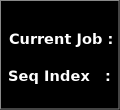
VISUALIZATION PUSeq  // 120x110
    Rectangle (0,0 371x118)
        OnMouseDown: CloseDialog Dialog=PUSeq, Result=None, NumpadKeypadSet=True
    Label (6,24 114x30), "Current Job :"
    Label (126,23 61x30)
    RoundedRectangle (121,24 235x29), "%s", tooltip "%s", text variable: HMI_GVL.sCurrentJob
        p4168582468: HMI_GVL.sCurrentJob
    RoundedRectangle (121,61 235x29), "%i", tooltip "%i", text variable: HMI_GVL.iSeqIndex
        p4168582468: HMI_GVL.iSeqIndex
    Label (5,61 121x30), "Seq Index :"
END_VISUALIZATION

(* stored: Version 1.1.0.1, ProductVersion 3.1.4024.12
   Visu PUSeq: Id {46e05c4c-b262-45b0-9067-450bb0be418c} *)
